// TIA Portal project "LearningFactory_4_0_24V_Task07_HighBayWarehouseHBW_V18" (V18)

(* hardware
DEVICE "ET 200SP-Station_1"  ET 200SP-Station
   slot 0: "Baugruppenträger_0"  Rack  6ES5 710-8MAx1
   slot 1: "PLC"  CPU 1512SP F-1 PN  6ES7 512-1SK01-0AB0  V2.8
      slot 32768: "PROFINET"  X1
   slot 2: "DO1+2"  DQ 16x24VDC/0.5A ST  6ES7 132-6BH01-0BA0  V0.0
      slot 1: "DO1+2"  DQ 16x24VDC/0.5A ST
   slot 3: "DO3+4"  DQ 16x24VDC/0.5A ST  6ES7 132-6BH01-0BA0  V0.0
      slot 1: "DO3+4"  DQ 16x24VDC/0.5A ST
   slot 4: "DO5+6"  DQ 16x24VDC/0.5A ST  6ES7 132-6BH01-0BA0  V0.0
      slot 1: "DO5+6"  DQ 16x24VDC/0.5A ST
   slot 5: "DO7-14"  DQ 4x24VDC/2A HS  6ES7 132-6BD20-0DA0  V2.0
      slot 1: "DO7-14"  DQ 4x24VDC/2A HS
   slot 6: "DO15-22"  DQ 4x24VDC/2A HS  6ES7 132-6BD20-0DA0  V2.0
      slot 1: "DO15-22"  DQ 4x24VDC/2A HS
   slot 7: "DO23-30"  DQ 4x24VDC/2A HS  6ES7 132-6BD20-0DA0  V2.0
      slot 1: "DO23-30"  DQ 4x24VDC/2A HS
   slot 8: "DI1+2"  DI 16x24VDC ST  6ES7 131-6BH01-0BA0  V0.0
      slot 1: "DI1+2"  DI 16x24VDC ST
   slot 9: "DI3+4"  DI 16x24VDC ST  6ES7 131-6BH01-0BA0  V0.0
      slot 1: "DI3+4"  DI 16x24VDC ST
   slot 10: "DI5"  DI 8x24VDC HS  6ES7 131-6BF00-0DA0  V1.0
      slot 1: "DI5"  DI 8x24VDC HS
   slot 11: "DI6"  DI 8x24VDC HS  6ES7 131-6BF00-0DA0  V1.0
      slot 1: "DI6"  DI 8x24VDC HS
   slot 12: "AI7-10"  AI 2xU ST  6ES7 134-6FB00-0BA1  V1.0
      slot 1: "AI7-10"  AI 2xU ST
   slot 13: "End"  Server module  6ES7 193-6PA00-0AA0  V1.1
      slot 1: "End"  Server module
   slot 127: "BA 2xRJ45"  BA 2xRJ45  6ES7 193-6AR00-0AA0  V0.0
      slot 32769: "Port_1"  6ES7 193-6AR00-0AA0
      slot 32770: "Port_2"  6ES7 193-6AR00-0AA0
*)

// ===== PLC "PLC"  CPU 1512SP F-1 PN =====

VAR_GLOBAL   // PLC tag table "Start_Stop"
   "IX_START" AT %I4.4 : Bool;
   "IX_STOP" AT %I4.6 : Bool;
END_VAR

VAR_GLOBAL   // PLC tag table "HBW - Automated High-Bay Warehouse"
   "IX_HBW_RefSwitchHorizontalAxis_I1" AT %I1.0 : Bool;
   "IX_HBW_LightBarrierInside_I2" AT %I1.1 : Bool;
   "IX_HBW_LightBarrierOutside_I3" AT %I1.2 : Bool;
   "IX_HBW_RefSwitchVerticalAxis_I4" AT %I1.3 : Bool;
   "IX_HBW_TrailSensor1Lower_A1" AT %I5.0 : Bool;
   "IX_HBW_TrailSensor2Upper_A2" AT %I5.4 : Bool;
   "IX_HBW_EncoderVerticalAxisImp1_B3" AT %I5.2 : Bool;
   "IX_HBW_EncoderVerticalAxisImp2_B4" AT %I5.6 : Bool;
   "IX_HBW_EncoderHorizontalAxisImp1_B1" AT %I5.1 : Bool;
   "IX_HBW_EncoderHorizontalAxisImp2_B2" AT %I5.5 : Bool;
   "IX_HBW_SwitchCantileverFront_I5" AT %I1.4 : Bool;
   "IX_HBW_SwitchCantileverBack_I6" AT %I1.5 : Bool;
   "QX_HBW_M1_ConveyorBeltForward_Q1" AT %Q1.0 : Bool;
   "QX_HBW_M1_ConveyorBeltBackward_Q2" AT %Q1.1 : Bool;
   "QX_HBW_M2_HorizontalTowardsRack_Q3" AT %Q1.2 : Bool;
   "QX_HBW_M2_HorizontalTowardsConveyorBelt_Q4" AT %Q1.3 : Bool;
   "QX_HBW_M3_VerticalAxisDownward_Q5" AT %Q1.4 : Bool;
   "QX_HBW_M3_VerticalAxisUpward_Q6" AT %Q1.5 : Bool;
   "QX_HBW_M4_CantileverForward_Q7" AT %Q1.6 : Bool;
   "QX_HBW_M4_CantileverBackward_Q8" AT %Q1.7 : Bool;
   "QW_HBW_PWM_ConveyorBelt_M1" AT %QW7 : Int;
   "QW_HBW_PWM_HorizontalAxis_M2" AT %QW9 : Int;
   "QW_HBW_PWM_VerticalAxis_M3" AT %QW11 : Int;
   "QW_HBW_PWM_Cantilever_M4" AT %QW13 : Int;
END_VAR

DATA_BLOCK "Task07_HighBayWarehouse_DB"   // DB5
{ S7_Optimized_Access := 'TRUE' }
VERSION : 0.1
// stored: InstanceOfName Task07_HighBayWarehouse
"Task07_HighBayWarehouse"
BEGIN
END_DATA_BLOCK

// folder: Positioning

DATA_BLOCK "Positioning"   // DB90
{ S7_Optimized_Access := 'TRUE' }
VERSION : 0.1
   VAR
      Axis_Horizontal : Struct
         Direction : Bool;
         Position : Int;
      END_STRUCT;
      Axis_Vertical : Struct
         Direction : Bool;
         Position : Int;
      END_STRUCT;
   END_VAR
BEGIN
END_DATA_BLOCK

DATA_BLOCK "FB_INC_DEC_DB_Horizontal"   // DB91
{ S7_Optimized_Access := 'TRUE' }
VERSION : 0.1
// stored: InstanceOfName FB_INC_DEC
"FB_INC_DEC"
BEGIN
END_DATA_BLOCK

DATA_BLOCK "FB_INC_DEC_DB_Vertikal"   // DB92
{ S7_Optimized_Access := 'TRUE' }
VERSION : 0.1
// stored: InstanceOfName FB_INC_DEC
"FB_INC_DEC"
BEGIN
END_DATA_BLOCK

// folder: (top level)

FUNCTION_BLOCK "Task07_HighBayWarehouse"   // FB5, SCL
{ S7_Optimized_Access := 'TRUE' }
VERSION : 0.1
   VAR_INPUT
      Start : Bool;
      Stop : Bool;
      RefSwitchHorizontalAxis : Bool;
      RefSwitchVerticalAxis : Bool;
      LightBarrierInside : Bool;
      LightBarrierOutside : Bool;
      SwitchCantileverFront : Bool;
      SwitchCantileverBack : Bool;
      PositionHorizontal : Int;
      PositionVertical : Int;
   END_VAR
   VAR_OUTPUT
      PWM_ConveyorBelt : Int;
      PWM_HorizontalAxis : Int;
      PWM_VerticalAxis : Int;
      PWM_Cantilever : Int;
   END_VAR
   VAR_IN_OUT
      M1_ConveyorBeltForward : Bool;
      M1_ConveyorBeltBackward : Bool;
      M2_HorizontalTowardsRack : Bool;
      M2_HorizontalTowardsConveyorBelt : Bool;
      M3_VerticalAxisDownward : Bool;
      M3_VerticalAxisUpward : Bool;
      M4_CantileverForward : Bool;
      M4_CantileverBackward : Bool;
   END_VAR
   VAR
      Step_number : Int;
      PositioningCounterVertical : Int;
      PositioningCounterRotate : Int;
      R_TRIG_PulseCountVertical : R_TRIG;
      R_TRIG_PulseCountRotate : R_TRIG;
      IEC_Timer_VacuumOn : TON_TIME;
      IEC_Timer_VacuumOff : TON_TIME;
   END_VAR
BEGIN

   // Reset sequencer with pushbutton STOP 
   // Rücksetzen der Schrittkette  mit Taster STOP
   IF #Stop THEN
       #Step_number := 0;
   END_IF;

   // Start sequencer with pushbutton START
   // Starten der Schrittkette  mit Taster START
   CASE #Step_number OF
       0:  // Initial step 1 / Initialschritt 1
           #M1_ConveyorBeltForward := FALSE;               //Conveyor forward off / Förderband vorwärts aus
           #M1_ConveyorBeltBackward := FALSE;             //Conveyor backward off / Förderband rückwärts aus
           #M2_HorizontalTowardsRack := FALSE;             //Horizontal axis towards rack off/ Horizontale Achse zum Lager aus    
           #M2_HorizontalTowardsConveyorBelt := FALSE;     //Horizontal axis towards conveyor off/ Horizontale Achse zum Förderband aus  
           #M3_VerticalAxisDownward := FALSE;              //Vertical axis down off / Vertikale Achse runterfahren aus
           #M3_VerticalAxisUpward := FALSE;                //Vertical axis up off/ Vertikale Achse hochfahren aus
           #M4_CantileverForward := FALSE;                 // Cantilever forward off / Ausleger vorwärts aus
           #M4_CantileverBackward := FALSE;                // Cantilever backward off / Ausleger rückwärts aus

           IF NOT #LightBarrierInside AND NOT #LightBarrierOutside
               AND #Start THEN
               #Step_number := #Step_number + 1;
           END_IF;

       1:  // Step 1 move back cantilever / Schritt 1 Ausleger einfahren
           #M4_CantileverBackward := TRUE;                // Cantilever backward / Ausleger rückwärts 

           IF #SwitchCantileverBack THEN
               #Step_number := #Step_number + 1;
           END_IF;

       2:  // Step 2 horizontal axis towards conveyor; vertical axis up;
           // Schritt 2 horizontale Achse zum Förderband; vertikale Achse nach oben
           #M4_CantileverBackward := FALSE;                // Cantilever backward off / Ausleger rückwärts aus
           #M2_HorizontalTowardsConveyorBelt := TRUE;     //Horizontal axis towards conveyor / Horizontale Achse zum Förderband 
           #M3_VerticalAxisUpward := TRUE;                //Vertical axis up / Vertikale Achse hochfahren 

           IF #RefSwitchHorizontalAxis THEN
               #M2_HorizontalTowardsConveyorBelt := FALSE;     //Horizontal axis towards conveyor off / Horizontale Achse Zum Förderband aus
           END_IF;
           IF #RefSwitchVerticalAxis THEN
               #M3_VerticalAxisUpward := FALSE;                //Vertical axis up off/ Vertikale Achse hochfahren aus
           END_IF;

           IF #RefSwitchHorizontalAxis AND #RefSwitchVerticalAxis THEN
               #Step_number := #Step_number + 1;
           END_IF;

       3:  // Step 3 horizontal axis and vertical axis towards position Rack A1;
           // Schritt 3 horizontale Achse und vertikale Achse zur Position Lager Rack A1
           #M2_HorizontalTowardsRack := TRUE;             //Horizontal axis towards rack / Horizontale Achse zum Lager 
           #M3_VerticalAxisDownward := TRUE;              //Vertical axis down / Vertikale Achse runterfahren 

           IF #PositionHorizontal >= 2920 THEN
               #M2_HorizontalTowardsRack := FALSE;              //Horizontal axis towards rack off/ Horizontale Achse zum Lager aus 
           END_IF;
           IF #PositionVertical >= 300 THEN
               #M3_VerticalAxisDownward := FALSE;               //Vertical axis down off / Vertikale Achse runterfahren aus
           END_IF;

           IF #PositionHorizontal >= 2920 AND #PositionVertical >= 300 THEN
               #Step_number := #Step_number + 1;
           END_IF;

       4:  // Step 4 cantilever forward /Schritt 4 Ausleger ausfahren
           #M4_CantileverForward := TRUE;             // Cantilever forward / Ausleger vorwärts 

           IF #SwitchCantileverFront THEN
               #Step_number := #Step_number + 1;
           END_IF;

       5:  // Step 5 vertical axis up lift box / Schritt 5 vertikale Achse hoch Box anheben
           #M4_CantileverForward := FALSE;             // Cantilever forward off / Ausleger vorwärts aus
           #M3_VerticalAxisUpward := TRUE;                //Vertical axis up / Vertikale Achse hochfahren 

           IF #PositionVertical <= 100 THEN
               #Step_number := #Step_number + 1;
           END_IF;

       6:  // Step 6 cantilever backward /Schritt 6 Ausleger einfahren
           #M3_VerticalAxisUpward := FALSE;                //Vertical axis up off / Vertikale Achse hochfahren aus
           #M4_CantileverBackward := TRUE;                // Cantilever backward / Ausleger rückwärts 

           IF #SwitchCantileverBack THEN
               #Step_number := #Step_number + 1;
           END_IF;

       7:  // Step 7 horizontal axis and vertical axis towards position conveyor;
           // Schritt 7 horizontale Achse und vertikale Achse zur Position Förderband
           #M4_CantileverBackward := FALSE;                // Cantilever backward off / Ausleger rückwärts aus
           #M2_HorizontalTowardsConveyorBelt := TRUE;     //Horizontal axis towards conveyor / Horizontale Achse zum Förderband 
           #M3_VerticalAxisDownward := TRUE;                //Vertical axis down / Vertikale Achse runterfahren 

           IF #PositionHorizontal <= 18 THEN
               #M2_HorizontalTowardsConveyorBelt := FALSE;     //Horizontal axis towards conveyor off / Horizontale Achse Zum Förderband aus
           END_IF;
           IF #PositionVertical >= 2600 THEN
               #M3_VerticalAxisDownward := FALSE;                //Vertical axis down off / Vertikale Achse runterfahren aus
           END_IF;

           IF #PositionHorizontal <= 18 AND #PositionVertical >= 2600 THEN
               #Step_number := #Step_number + 1;
           END_IF;

       8:  // Step 8 cantilever forward /Schritt 8 Ausleger ausfahren
           #M4_CantileverForward := TRUE;             // Cantilever forward / Ausleger vorwärts 

           IF #SwitchCantileverFront THEN
               #Step_number := #Step_number + 1;
           END_IF;

       9:  // Step 9 vertical axis down deposit box / Schritt 9 vertikale Achse runter Box ablegen
           #M4_CantileverForward := FALSE;             // Cantilever forward off / Ausleger vorwärts aus
           #M3_VerticalAxisDownward := TRUE;                //Vertical axis down / Vertikale Achse runterfahren 

           IF #LightBarrierInside AND #PositionVertical >= 2800 THEN
               #Step_number := #Step_number + 1;
           END_IF;

       10: // Step 6 cantilever backward; conveyor forward
           // Schritt 6 Ausleger einfahren; Förderband vorwärts
           #M3_VerticalAxisDownward := FALSE;             //Vertical axis down off / Vertikale Achse runterfahren aus
           #M4_CantileverBackward := TRUE;                // Cantilever backward / Ausleger rückwärts 
           #M1_ConveyorBeltForward := TRUE;               //Conveyor forward / Förderband vorwärts

           IF #SwitchCantileverBack THEN
               #M4_CantileverBackward := FALSE;                // Cantilever backward off / Ausleger rückwärts aus
           END_IF;
           IF #LightBarrierOutside THEN
               #M1_ConveyorBeltForward := FALSE;               //Conveyor forward off / Förderband vorwärts aus
           END_IF;

           IF #SwitchCantileverBack AND #LightBarrierOutside THEN
               #Step_number := 0;
          END_IF;

       ELSE  // Statement section ELSE
           ;
   END_CASE;


   //Permanent Instructions

   //Pulse width modulation control for conveyor
   //Pulsweitenmodulation für Drehtisch
   IF #M1_ConveyorBeltForward OR #M1_ConveyorBeltBackward
   THEN
       #PWM_ConveyorBelt := 500;
   ELSE
       #PWM_ConveyorBelt := 0;
   END_IF;

   //Pulse width modulation control for linear axle vacuum gripper
   //Pulsweitenmodulation für Linearachse Vakuumgreifer
   IF #M2_HorizontalTowardsRack OR #M2_HorizontalTowardsConveyorBelt
   THEN
       #PWM_HorizontalAxis := 500;
   ELSE
       #PWM_HorizontalAxis := 0;
   END_IF;

   //Pulse width modulation control for linear axle vacuum gripper
   //Pulsweitenmodulation für Linearachse Vakuumgreifer
   IF #M3_VerticalAxisDownward OR #M3_VerticalAxisUpward
   THEN
       #PWM_VerticalAxis := 500;
   ELSE
       #PWM_VerticalAxis := 0;
   END_IF;

   //Pulse width modulation control for linear axle vacuum gripper
   //Pulsweitenmodulation für Linearachse Vakuumgreifer
   IF #M4_CantileverForward OR #M4_CantileverBackward
   THEN
       #PWM_Cantilever := 500;
   ELSE
       #PWM_Cantilever := 0;
   END_IF;
END_FUNCTION_BLOCK

ORGANIZATION_BLOCK "Main"   // OB1, SCL, ProgramCycle
TITLE = "Main Program Sweep (Cycle)"
{ S7_Optimized_Access := 'TRUE' }
VERSION : 0.1
   VAR_INPUT
      Initial_Call : Bool;   // Initial call of this OB
      Remanence : Bool;   // =True, if remanent data are available
   END_VAR
BEGIN


   // Call subroutine HighBayWarehouse
   // Aufruf Unterprogramm HighBayWarehouse

   "Task07_HighBayWarehouse_DB"(Start:="IX_START",
                                Stop:= NOT "IX_STOP",
                                RefSwitchHorizontalAxis:="IX_HBW_RefSwitchHorizontalAxis_I1",
                                RefSwitchVerticalAxis:="IX_HBW_RefSwitchVerticalAxis_I4",
                                LightBarrierInside:= NOT "IX_HBW_LightBarrierInside_I2",
                                LightBarrierOutside:= NOT "IX_HBW_LightBarrierOutside_I3",
                                SwitchCantileverFront:="IX_HBW_SwitchCantileverFront_I5",
                                SwitchCantileverBack:="IX_HBW_SwitchCantileverBack_I6",
                                PositionHorizontal:="Positioning".Axis_Horizontal.Position,
                                PositionVertical:="Positioning".Axis_Vertical.Position,
                                PWM_ConveyorBelt=>"QW_HBW_PWM_ConveyorBelt_M1",
                                PWM_HorizontalAxis=>"QW_HBW_PWM_HorizontalAxis_M2",
                                PWM_VerticalAxis=>"QW_HBW_PWM_VerticalAxis_M3",
                                PWM_Cantilever=>"QW_HBW_PWM_Cantilever_M4",
                                M1_ConveyorBeltForward:="QX_HBW_M1_ConveyorBeltForward_Q1",
                                M1_ConveyorBeltBackward:="QX_HBW_M1_ConveyorBeltBackward_Q2",
                                M2_HorizontalTowardsRack:="QX_HBW_M2_HorizontalTowardsRack_Q3",
                                M2_HorizontalTowardsConveyorBelt:="QX_HBW_M2_HorizontalTowardsConveyorBelt_Q4",
                                M3_VerticalAxisDownward:="QX_HBW_M3_VerticalAxisDownward_Q5",
                                M3_VerticalAxisUpward:="QX_HBW_M3_VerticalAxisUpward_Q6",
                                M4_CantileverForward:="QX_HBW_M4_CantileverForward_Q7",
                                M4_CantileverBackward:="QX_HBW_M4_CantileverBackward_Q8");
END_ORGANIZATION_BLOCK

// folder: Positioning

FUNCTION_BLOCK "FB_INC_DEC"   // FB9, SCL
TITLE = position with encoder
{ S7_Optimized_Access := 'TRUE' }
VERSION : 0.1
   VAR_INPUT
      inx_CHa : Bool := false;   // Encoder impulse 2 channel a / Encoderimpulse 2 Kanal a
      inx_CHb : Bool := false;   // Encoder impulse 1 channel b / / Encoderimpulse 1 Kanal b
      inx_RST : Bool := False;   // Reference switch / Referenzpunkt
      ini_Ref_val : Int := 0;   // Reference value / Referenzwert
   END_VAR
   VAR_OUTPUT
      outx_dir : Bool := false;   // direction / Richtung
      outi_cnt : Int := 0;   // position / Position
   END_VAR
   VAR
      lx_edgea : Bool := False;
      lx_clka : Bool;
      lx_clkb : Bool;
      lx_edgeb : Bool;
      lx_axb : Bool;
      lx_dir : Bool;
      li_cnt : Int;
   END_VAR
BEGIN

   #lx_axb := #inx_CHa XOR #inx_CHb;
   (* create pulses for channel a *)
   #lx_clka := #inx_CHa XOR #lx_edgea;
   #lx_edgea := #inx_CHa;
   (* create pulses for channel b *)
   #lx_clkb := #inx_CHb XOR #lx_edgeb;
   #lx_edgeb := #inx_CHb;
   (* create pulses for both channels *)
   #lx_clka := #lx_clka OR #lx_clkb;
   (* set the direction output *)
   IF #lx_axb AND #lx_clka THEN
       #lx_dir := TRUE;
   END_IF;
   IF #lx_axb AND #lx_clkb THEN
       #lx_dir := FALSE;
   END_IF;
   (* increment or decrement the counter *)
   IF #lx_clka AND #lx_dir THEN
       #li_cnt := #li_cnt + 1;
   END_IF;
   IF #lx_clka AND NOT #lx_dir THEN
       #li_cnt := #li_cnt - 1;
   END_IF;
   (* reset the counter if rst active *)
   IF #inx_RST THEN
       #li_cnt := #ini_Ref_val;
   END_IF;
   #outx_dir := #lx_dir;
   #outi_cnt := #li_cnt;
END_FUNCTION_BLOCK

ORGANIZATION_BLOCK "Cyclic interrupt"   // OB30, SCL, CyclicInterrupt
{ S7_Optimized_Access := 'TRUE' }
VERSION : 0.1
   VAR_INPUT
      Initial_Call : Bool;   // Initial call of this OB
      Event_Count : Int;   // Events discarded
   END_VAR
   VAR_TEMP
      li_Return_LDT : Int;
   END_VAR
BEGIN

   // Call FB increment axis -> get direction and position horizontal
   // Aufruf FB Inkremente Achse -> Richtung und Position horizontal
   "FB_INC_DEC_DB_Horizontal"(inx_CHa := "IX_HBW_EncoderHorizontalAxisImp2_B2",
               inx_CHb := "IX_HBW_EncoderHorizontalAxisImp1_B1",
               inx_RST := "IX_HBW_RefSwitchHorizontalAxis_I1",
               ini_Ref_val := 0,
               outx_dir=>"Positioning".Axis_Horizontal.Direction,
               outi_cnt=>"Positioning".Axis_Horizontal.Position);

   // Call FB increment axis -> get direction and position vertical
   // Aufruf FB Inkremente Achse -> Richtung und Position vertikal
   "FB_INC_DEC_DB_Vertikal"(inx_CHa := "IX_HBW_EncoderVerticalAxisImp1_B3",
               inx_CHb := "IX_HBW_EncoderVerticalAxisImp2_B4",
               inx_RST := "IX_HBW_RefSwitchVerticalAxis_I4",
               ini_Ref_val := 0,
               outx_dir=>"Positioning".Axis_Vertical.Direction,
               outi_cnt=>"Positioning".Axis_Vertical.Position);
END_ORGANIZATION_BLOCK